Staubli VAL3: feedbackStatus.pgx

public program feedbackStatus(num x_nOutConnFlag)
begin

  // update connection status on port 11002 (feedback server)

  switch x_nOutConnFlag
    case -1
      userPageSet("uxMonitor", "lblFeedbackState", "innerHTML", "connection lost")
    break
    case 0
      userPageSet("uxMonitor", "lblFeedbackState", "innerHTML", "not connected")
    break
    case 1
      userPageSet("uxMonitor", "lblFeedbackState", "innerHTML", "connected")
    break
    default
      userPageSet("uxMonitor", "lblFeedbackState", "innerHTML", "not connected")
    break
  endSwitch

end
